(* Logix 5000 project; controller DUNEW2PLC1 vendor 1 type 14 code 221 rev 33.11; software revision 33.00; part 2 of 4 *)
(* tags used below, declared in another part *)
   LatchingTimeoutCounter : COUNTER;   // When you enter state 6 or 7, start counting seconds
   TimeoutTimer1 : TIMER;
   TimeoutTimer2 : TIMER;
   accel_xy : REAL;   // Tangential acceleration of the winding head in xy-plane
   ACTUATOR_POS : DINT;
   ALL_EOT_GOOD : BOOL;
   APA_IS_VERTICAL : BOOL;
   blink_off : TIMER;
   blink_on : TIMER;
   ERROR_CODE : DINT;
   FRAME_LOC_FT_BTM : BOOL;
   FRAME_LOC_FT_MID : BOOL;
   FRAME_LOC_FT_TOP : BOOL;
   FRAME_LOC_HD_BTM : BOOL;
   FRAME_LOC_HD_MID : BOOL;
   FRAME_LOC_HD_TOP : BOOL;
   HEAD_POS : DINT;
   INIT_DONE : BOOL;
   MACHINE_SW_STAT : BOOL[32];
   MAS : BOOL;   // Motion Axis Stop
   MASTER_Z_GO : BOOL;
   MCCD_X_Y_Axis : MOTION_INSTRUCTION;
   MCCD_X_Y_Axis1 : MOTION_INSTRUCTION;
   MINUS_X_EOT : BOOL;
   MINUS_Y_EOT : BOOL;
   MOVE_TYPE : INT;   // 0 = No Move 1 = XY JOG 2 = XY Plane Move 3 = Z JOG 4 = Z Axis Move 5 = Toggle Latch Actuator 6 = Home the Latch Actuator
   NEXTSTATE : DINT;
   PLUS_X_EOT : BOOL;
   PLUS_Y_EOT : BOOL;
   ResetPB : BOOL;
   Safety_Tripped_S : BOOL;
   SLS_speed : DINT;
   speed_regulator_switch : BOOL;   // This is our "enable safe speed" switch, repurposed to switch the speed regulator
   STATE : DINT;   // CURRENT State Machine State
   T01 : TIMER;
   tension : ALIAS FOR Local:4:I.Ch01.Data;   // wire tension (N)
   TENSION_ON_SWITCH : BOOL;
   v_xy : REAL;   // velocity of winding head in xy plane
   v_xyz : REAL;   // Velocity of winding head in xyz space
   wire_break_proxy : BOOL;
   wire_break_tension : REAL;
   X_axis : AXIS_CIP_DRIVE;
   X_Axis_SLS : SAFELY_LIMITED_SPEED;
   X_DIR : DINT;
   X_PARKED : BOOL;
   X_POSITION : ALIAS FOR POSITION[0,0];
   X_SPEED : REAL;
   X_XFER_OK : BOOL;   // If at the head, check head support arms. Same for foot
   X_Y : COORDINATE_SYSTEM;
   XY_ACCELERATION : REAL;   // Maximum positive acceleration for position move.
   XY_DECELERATION : REAL;   // Maximum negative acceleration for position move.
   XY_DECELERATION_SLS : REAL;
   XY_SPEED : REAL;   // Maximum velocity for position move.
   XY_SPEED_REQ : REAL;   // XY Requested speed copy of XY_Speed to be used for MCLM and MCCD in MoveXY
   Y_axis : AXIS_CIP_DRIVE;
   Y_DIR : DINT;
   Y_MOUNT_XFER_OK : BOOL;
   Y_POSITION : ALIAS FOR POSITION[0,1];
   Y_SPEED : REAL;
   Y_XFER_OK : BOOL;
   Y_Xfer_Window_Btm : BOOL;
   Y_Xfer_Window_Mid : BOOL;
   Y_Xfer_Window_Top : BOOL;
   Z_axis : AXIS_CIP_DRIVE;
   Z_EOT : BOOL;
   Z_EXTENDED : BOOL;
   Z_FIXED_LATCHED : BOOL;
   Z_FIXED_PRESENT : BOOL;
   Z_RETRACTED : BOOL;
   Z_STAGE_LATCHED : BOOL;
   Z_STAGE_PRESENT : BOOL;   // Winding head is on the Z-arm
(* Latch_UnLatch_State_6_7_8, continued *)

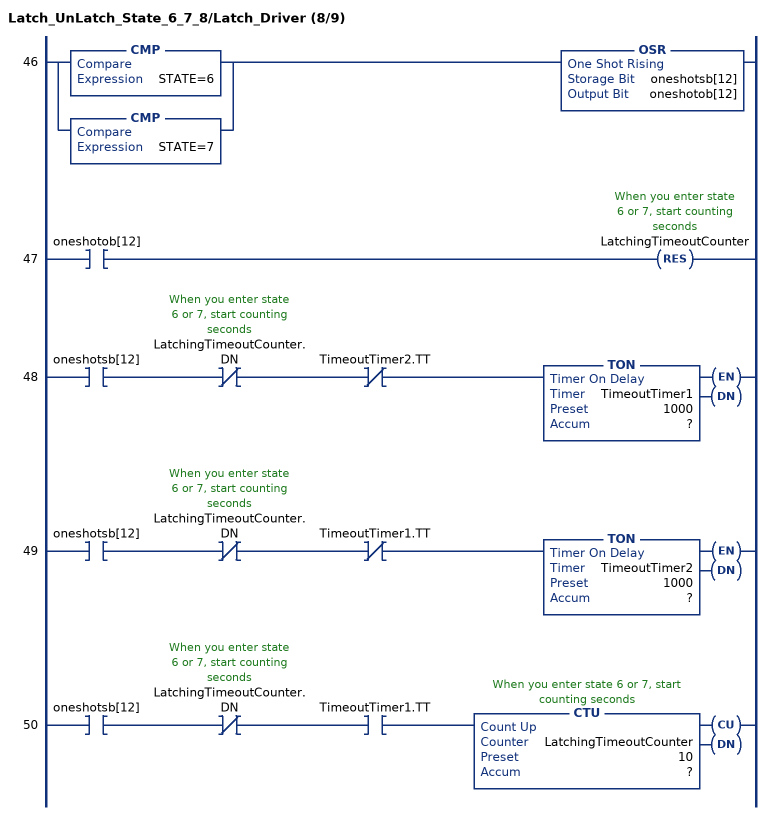
   [picture p24: Latch_UnLatch_State_6_7_8/Latch_Driver rungs 46-50]
   46: [CMP(STATE=6) ,CMP(STATE=7) ]OSR(oneshotsb[12],oneshotob[12]);
   47: XIC(oneshotob[12])RES(LatchingTimeoutCounter);
   48: XIC(oneshotsb[12])XIO(LatchingTimeoutCounter.DN)XIO(TimeoutTimer2.TT)TON(TimeoutTimer1,?,?);
   49: XIC(oneshotsb[12])XIO(LatchingTimeoutCounter.DN)XIO(TimeoutTimer1.TT)TON(TimeoutTimer2,?,?);
   50: XIC(oneshotsb[12])XIO(LatchingTimeoutCounter.DN)XIC(TimeoutTimer1.TT)CTU(LatchingTimeoutCounter,?,?);
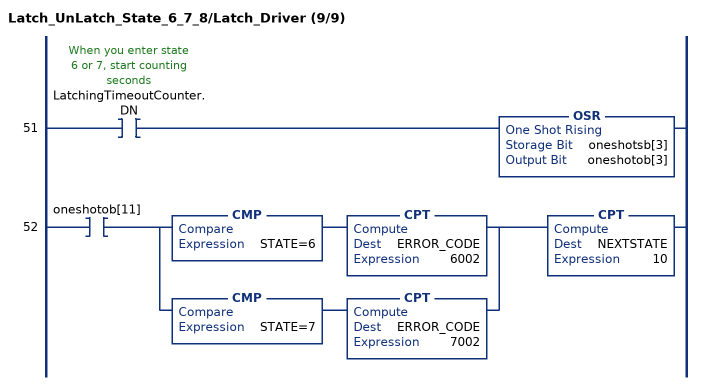
   51: XIC(LatchingTimeoutCounter.DN)OSR(oneshotsb[3],oneshotob[3]);
   52: XIC(oneshotob[11])[CMP(STATE=6) CPT(ERROR_CODE,6002) ,CMP(STATE=7) CPT(ERROR_CODE,7002) ]CPT(NEXTSTATE,10);
END_ROUTINE
END_PROGRAM

PROGRAM MainProgram   (* main routine MainRoutine *)
VAR
   Current_x : REAL := 0.0057; {access Read Only}
   Current_y : DINT; {access Read Only}
   oneshotob : BOOL[32];
   oneshotsb : BOOL[32] := ([4] := 1, [7] := 1);
   STATE2_IND : BOOL; {access Read Only}
   STATE3_IND : BOOL; {access Read Only}
   X_AXIS_STAT : MOTION_INSTRUCTION[32] := ([0].FLAGS := 33554432, [1].FLAGS := 33554432, [2].FLAGS := 33554432);
   XY_AXIS_STAT : MOTION_INSTRUCTION[32] := ([0].FLAGS := 33554432, [1].FLAGS := 33554432, [2].FLAGS := 536870912, [2].DN := 1, [3].FLAGS := 536870912, [3].DN := 1, [4].FLAGS := 704643072, [4].DN := 1, [4].PC := 1, [5].FLAGS := 704643072, [5].DN := 1, [5].PC := 1, [6].FLAGS := 33554432);
   XY_POS_LOCK_STAT : BOOL; {access Read Only}
   XY_SERVO_ON : BOOL; {access Read Only}
   Y_AXIS_STAT : MOTION_INSTRUCTION[32] := ([0].FLAGS := 33554432, [1].FLAGS := 33554432, [2].FLAGS := 33554432);
   Z_RETRACTED_1A : BOOL := 1; {access Read Only}
   Z_RETRACTED_1B : BOOL := 1; {access Read Only}
   Z_RETRACTED_2A : BOOL := 1; {access Read Only}
   Z_RETRACTED_2B : BOOL := 1; {access Read Only}
END_VAR

ROUTINE MainRoutine   (* ladder *)
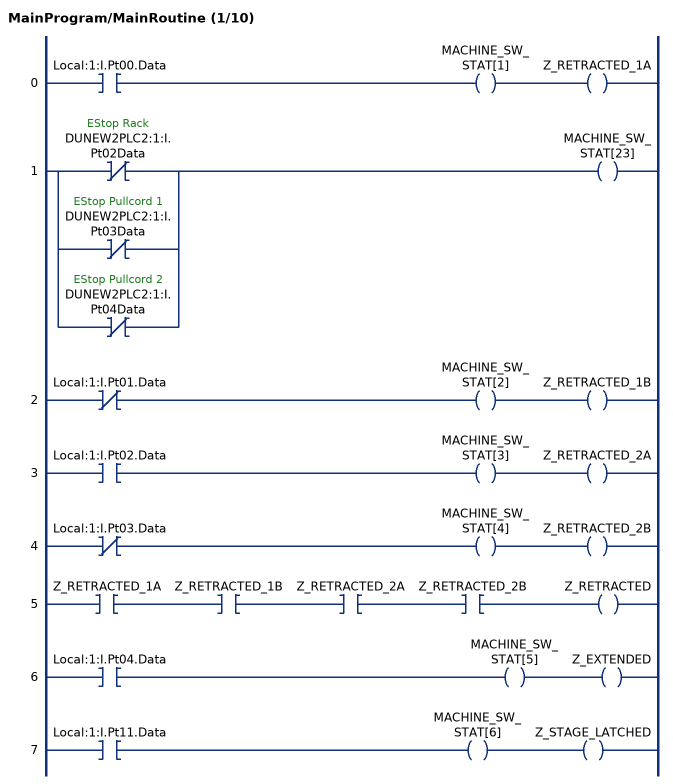
   0: XIC(Local:1:I.Pt00.Data)OTE(MACHINE_SW_STAT[1])OTE(Z_RETRACTED_1A);
   1: [XIO(DUNEW2PLC2:1:I.Pt02Data) ,[XIO(DUNEW2PLC2:1:I.Pt03Data) ,XIO(DUNEW2PLC2:1:I.Pt04Data) ] ]OTE(MACHINE_SW_STAT[23]);
   2: XIO(Local:1:I.Pt01.Data)OTE(MACHINE_SW_STAT[2])OTE(Z_RETRACTED_1B);
   3: XIC(Local:1:I.Pt02.Data)OTE(MACHINE_SW_STAT[3])OTE(Z_RETRACTED_2A);
   4: XIO(Local:1:I.Pt03.Data)OTE(MACHINE_SW_STAT[4])OTE(Z_RETRACTED_2B);
   5: XIC(Z_RETRACTED_1A)XIC(Z_RETRACTED_1B)XIC(Z_RETRACTED_2A)XIC(Z_RETRACTED_2B)OTE(Z_RETRACTED);
   6: XIC(Local:1:I.Pt04.Data)OTE(MACHINE_SW_STAT[5])OTE(Z_EXTENDED);
   7: XIC(Local:1:I.Pt11.Data)OTE(MACHINE_SW_STAT[6])OTE(Z_STAGE_LATCHED);
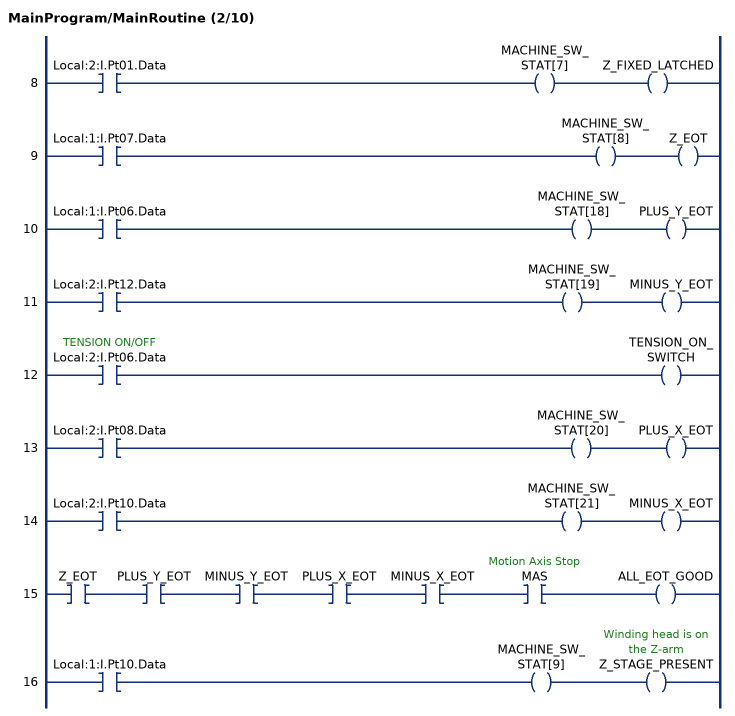
   8: XIC(Local:2:I.Pt01.Data)OTE(MACHINE_SW_STAT[7])OTE(Z_FIXED_LATCHED);
   9: XIC(Local:1:I.Pt07.Data)OTE(MACHINE_SW_STAT[8])OTE(Z_EOT);
   10: XIC(Local:1:I.Pt06.Data)OTE(MACHINE_SW_STAT[18])OTE(PLUS_Y_EOT);
   11: XIC(Local:2:I.Pt12.Data)OTE(MACHINE_SW_STAT[19])OTE(MINUS_Y_EOT);
   12: XIC(Local:2:I.Pt06.Data)OTE(TENSION_ON_SWITCH);
   13: XIC(Local:2:I.Pt08.Data)OTE(MACHINE_SW_STAT[20])OTE(PLUS_X_EOT);
   14: XIC(Local:2:I.Pt10.Data)OTE(MACHINE_SW_STAT[21])OTE(MINUS_X_EOT);
   15: XIC(Z_EOT)XIC(PLUS_Y_EOT)XIC(MINUS_Y_EOT)XIC(PLUS_X_EOT)XIC(MINUS_X_EOT)XIC(MAS)OTE(ALL_EOT_GOOD);
   16: XIC(Local:1:I.Pt10.Data)OTE(MACHINE_SW_STAT[9])OTE(Z_STAGE_PRESENT);
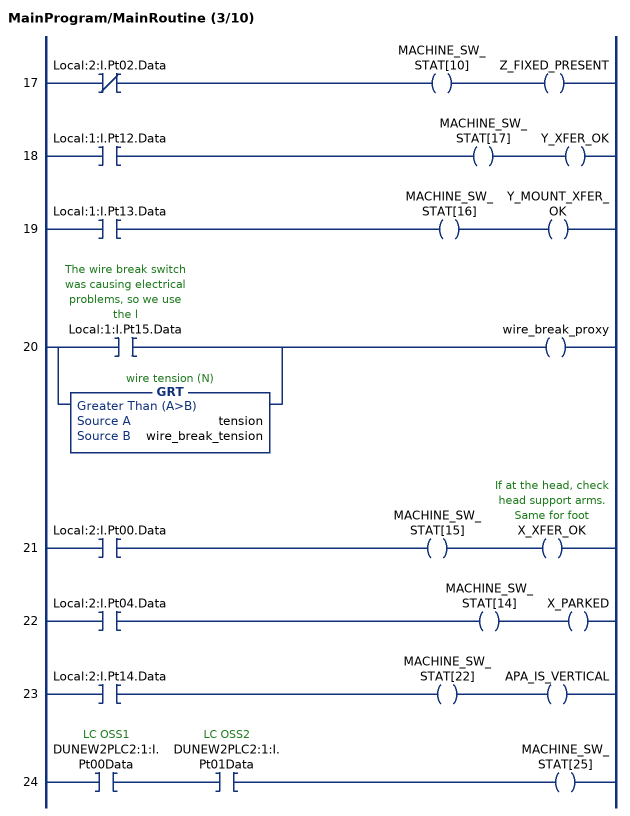
   17: XIO(Local:2:I.Pt02.Data)OTE(MACHINE_SW_STAT[10])OTE(Z_FIXED_PRESENT);
   18: XIC(Local:1:I.Pt12.Data)OTE(MACHINE_SW_STAT[17])OTE(Y_XFER_OK);
   19: XIC(Local:1:I.Pt13.Data)OTE(MACHINE_SW_STAT[16])OTE(Y_MOUNT_XFER_OK);
   20: [XIC(Local:1:I.Pt15.Data) ,GRT(tension,wire_break_tension) ]OTE(wire_break_proxy);
   21: XIC(Local:2:I.Pt00.Data)OTE(MACHINE_SW_STAT[15])OTE(X_XFER_OK);
   22: XIC(Local:2:I.Pt04.Data)OTE(MACHINE_SW_STAT[14])OTE(X_PARKED);
   23: XIC(Local:2:I.Pt14.Data)OTE(MACHINE_SW_STAT[22])OTE(APA_IS_VERTICAL);
   24: XIC(DUNEW2PLC2:1:I.Pt00Data)XIC(DUNEW2PLC2:1:I.Pt01Data)OTE(MACHINE_SW_STAT[25]);
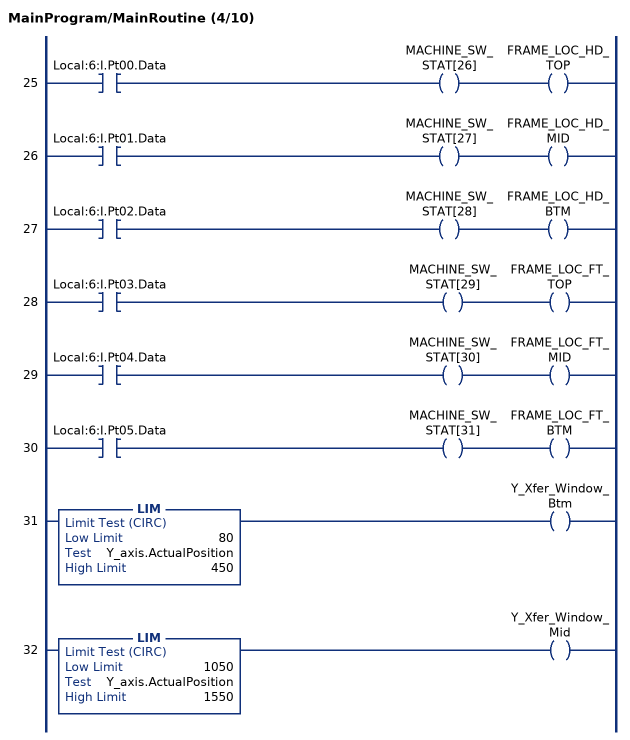
   25: XIC(Local:6:I.Pt00.Data)OTE(MACHINE_SW_STAT[26])OTE(FRAME_LOC_HD_TOP);
   26: XIC(Local:6:I.Pt01.Data)OTE(MACHINE_SW_STAT[27])OTE(FRAME_LOC_HD_MID);
   27: XIC(Local:6:I.Pt02.Data)OTE(MACHINE_SW_STAT[28])OTE(FRAME_LOC_HD_BTM);
   28: XIC(Local:6:I.Pt03.Data)OTE(MACHINE_SW_STAT[29])OTE(FRAME_LOC_FT_TOP);
   29: XIC(Local:6:I.Pt04.Data)OTE(MACHINE_SW_STAT[30])OTE(FRAME_LOC_FT_MID);
   30: XIC(Local:6:I.Pt05.Data)OTE(MACHINE_SW_STAT[31])OTE(FRAME_LOC_FT_BTM);
   31: LIM(80,Y_axis.ActualPosition,450)OTE(Y_Xfer_Window_Btm);
   32: LIM(1050,Y_axis.ActualPosition,1550)OTE(Y_Xfer_Window_Mid);
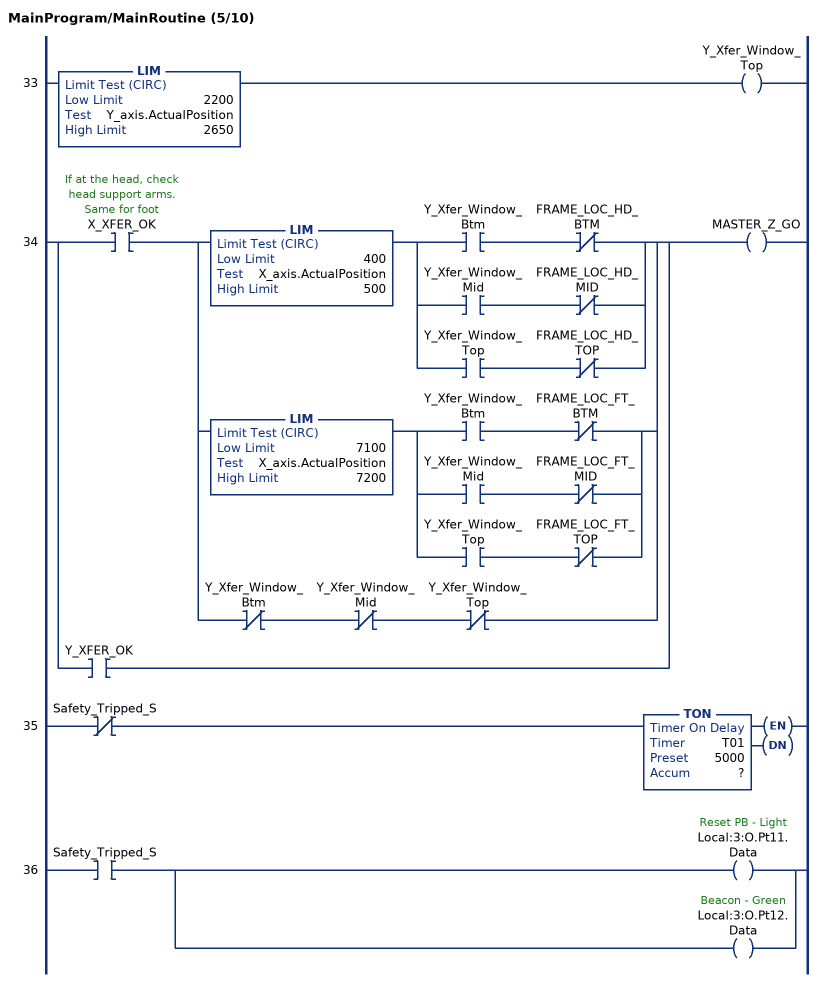
   33: LIM(2200,Y_axis.ActualPosition,2650)OTE(Y_Xfer_Window_Top);
   34: [XIC(X_XFER_OK) [LIM(400,X_axis.ActualPosition,500) [XIC(Y_Xfer_Window_Btm) XIO(FRAME_LOC_HD_BTM) ,XIC(Y_Xfer_Window_Mid) XIO(FRAME_LOC_HD_MID) ,XIC(Y_Xfer_Window_Top) XIO(FRAME_LOC_HD_TOP) ] ,LIM(7100,X_axis.ActualPosition,7200) [XIC(Y_Xfer_Window_Btm) XIO(FRAME_LOC_FT_BTM) ,XIC(Y_Xfer_Window_Mid) XIO(FRAME_LOC_FT_MID) ,XIC(Y_Xfer_Window_Top) XIO(FRAME_LOC_FT_TOP) ] ,XIO(Y_Xfer_Window_Btm) XIO(Y_Xfer_Window_Mid) XIO(Y_Xfer_Window_Top) ] ,XIC(Y_XFER_OK) ]OTE(MASTER_Z_GO);
   35: XIO(Safety_Tripped_S)TON(T01,?,?);
   36: XIC(Safety_Tripped_S)[OTE(Local:3:O.Pt11.Data) ,OTE(Local:3:O.Pt12.Data) ];
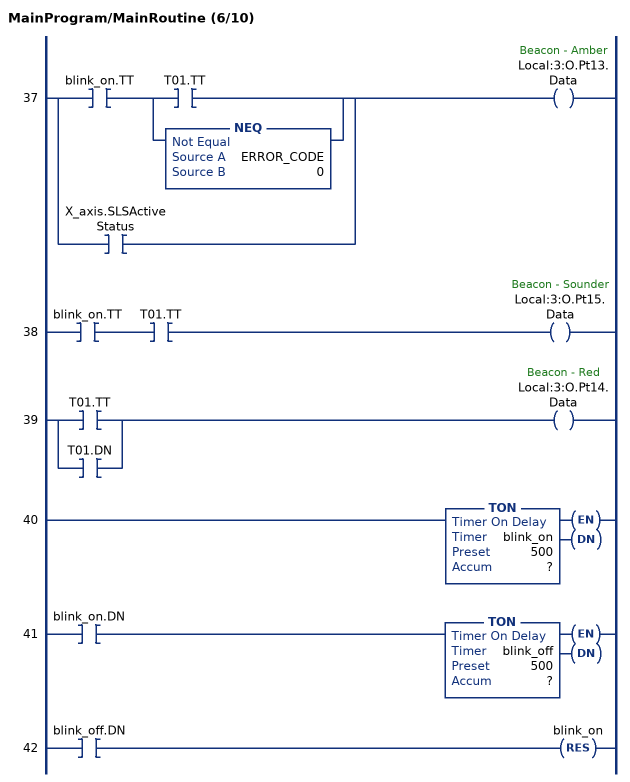
   37: [XIC(blink_on.TT) [XIC(T01.TT) ,NEQ(ERROR_CODE,0) ] ,XIC(X_axis.SLSActiveStatus) ]OTE(Local:3:O.Pt13.Data);
   38: XIC(blink_on.TT)XIC(T01.TT)OTE(Local:3:O.Pt15.Data);
   39: [XIC(T01.TT) ,XIC(T01.DN) ]OTE(Local:3:O.Pt14.Data);
   40: TON(blink_on,?,?);
   41: XIC(blink_on.DN)TON(blink_off,?,?);
   42: XIC(blink_off.DN)RES(blink_on);
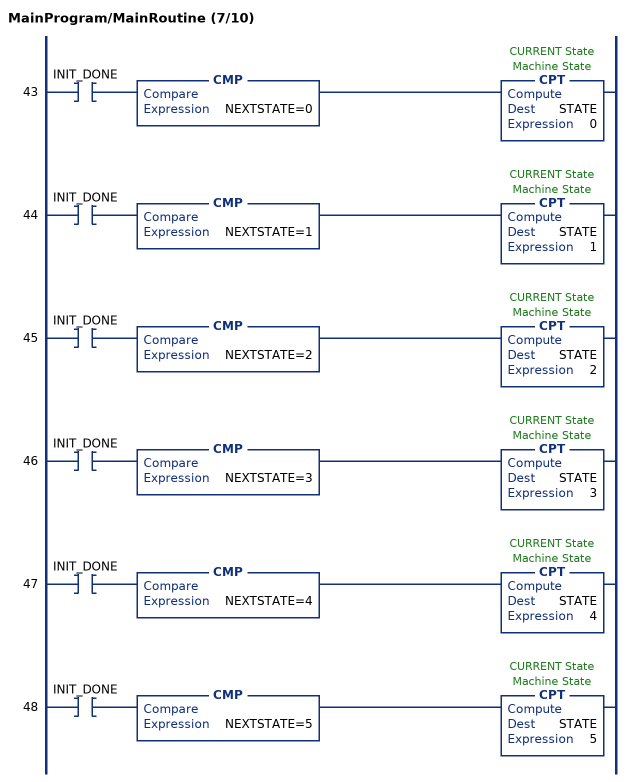
   43: XIC(INIT_DONE)CMP(NEXTSTATE=0)CPT(STATE,0);
   44: XIC(INIT_DONE)CMP(NEXTSTATE=1)CPT(STATE,1);
   45: XIC(INIT_DONE)CMP(NEXTSTATE=2)CPT(STATE,2);
   46: XIC(INIT_DONE)CMP(NEXTSTATE=3)CPT(STATE,3);
   47: XIC(INIT_DONE)CMP(NEXTSTATE=4)CPT(STATE,4);
   48: XIC(INIT_DONE)CMP(NEXTSTATE=5)CPT(STATE,5);
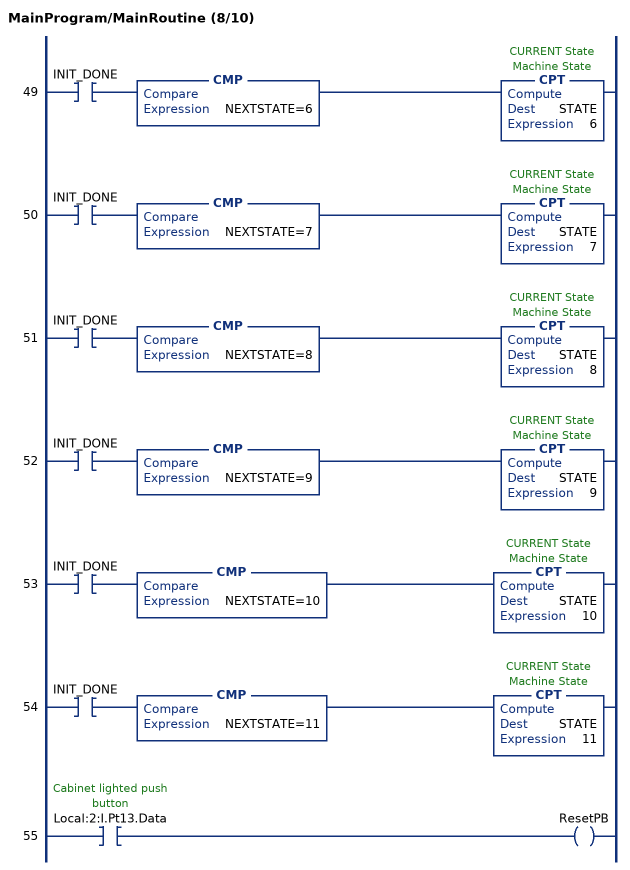
   49: XIC(INIT_DONE)CMP(NEXTSTATE=6)CPT(STATE,6);
   50: XIC(INIT_DONE)CMP(NEXTSTATE=7)CPT(STATE,7);
   51: XIC(INIT_DONE)CMP(NEXTSTATE=8)CPT(STATE,8);
   52: XIC(INIT_DONE)CMP(NEXTSTATE=9)CPT(STATE,9);
   53: XIC(INIT_DONE)CMP(NEXTSTATE=10)CPT(STATE,10);
   54: XIC(INIT_DONE)CMP(NEXTSTATE=11)CPT(STATE,11);
   55: XIC(Local:2:I.Pt13.Data)OTE(ResetPB);
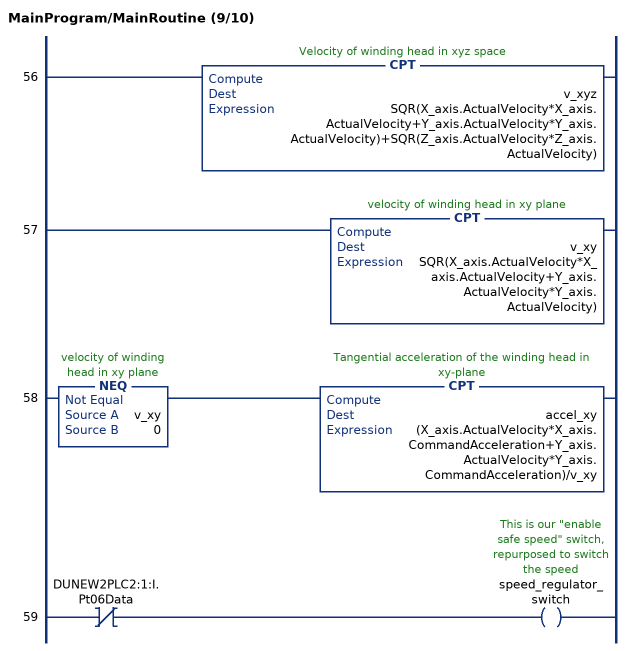
   56: CPT(v_xyz,SQR(X_axis.ActualVelocity*X_axis.ActualVelocity+Y_axis.ActualVelocity*Y_axis.ActualVelocity)+SQR(Z_axis.ActualVelocity*Z_axis.ActualVelocity));
   57: CPT(v_xy,SQR(X_axis.ActualVelocity*X_axis.ActualVelocity+Y_axis.ActualVelocity*Y_axis.ActualVelocity));
   58: NEQ(v_xy,0)CPT(accel_xy,(X_axis.ActualVelocity*X_axis.CommandAcceleration+Y_axis.ActualVelocity*Y_axis.CommandAcceleration)/v_xy);
   59: XIO(DUNEW2PLC2:1:I.Pt06Data)OTE(speed_regulator_switch);
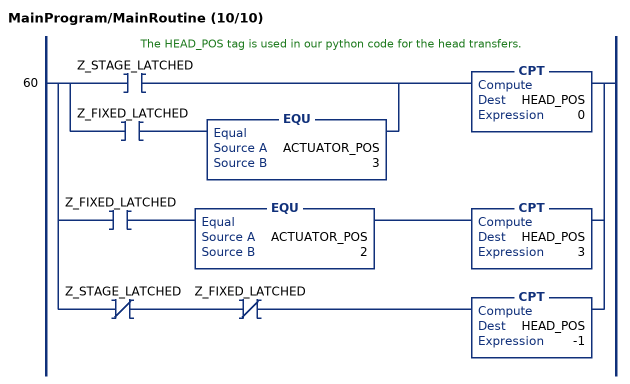
   // The HEAD_POS tag is used in our python code for the head transfers.
   60: [[XIC(Z_STAGE_LATCHED) ,XIC(Z_FIXED_LATCHED) EQU(ACTUATOR_POS,3) ] CPT(HEAD_POS,0) ,XIC(Z_FIXED_LATCHED) EQU(ACTUATOR_POS,2) CPT(HEAD_POS,3) ,XIO(Z_STAGE_LATCHED) XIO(Z_FIXED_LATCHED) CPT(HEAD_POS,-1) ];
END_ROUTINE

ROUTINE MoveXY   (* ladder *)
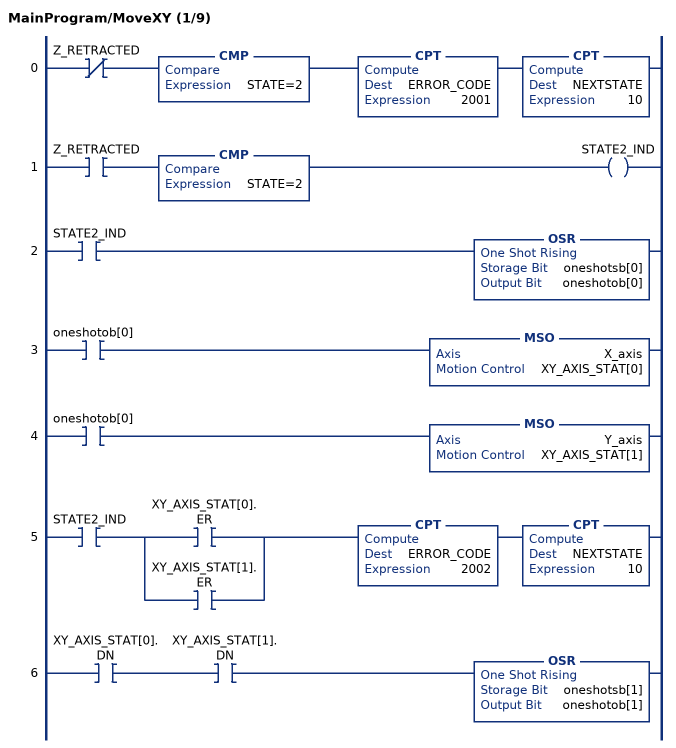
   0: XIO(Z_RETRACTED)CMP(STATE=2)CPT(ERROR_CODE,2001)CPT(NEXTSTATE,10);
   1: XIC(Z_RETRACTED)CMP(STATE=2)OTE(STATE2_IND);
   2: XIC(STATE2_IND)OSR(oneshotsb[0],oneshotob[0]);
   3: XIC(oneshotob[0])MSO(X_axis,XY_AXIS_STAT[0]);
   4: XIC(oneshotob[0])MSO(Y_axis,XY_AXIS_STAT[1]);
   5: XIC(STATE2_IND)[XIC(XY_AXIS_STAT[0].ER) ,XIC(XY_AXIS_STAT[1].ER) ]CPT(ERROR_CODE,2002)CPT(NEXTSTATE,10);
   6: XIC(XY_AXIS_STAT[0].DN)XIC(XY_AXIS_STAT[1].DN)OSR(oneshotsb[1],oneshotob[1]);
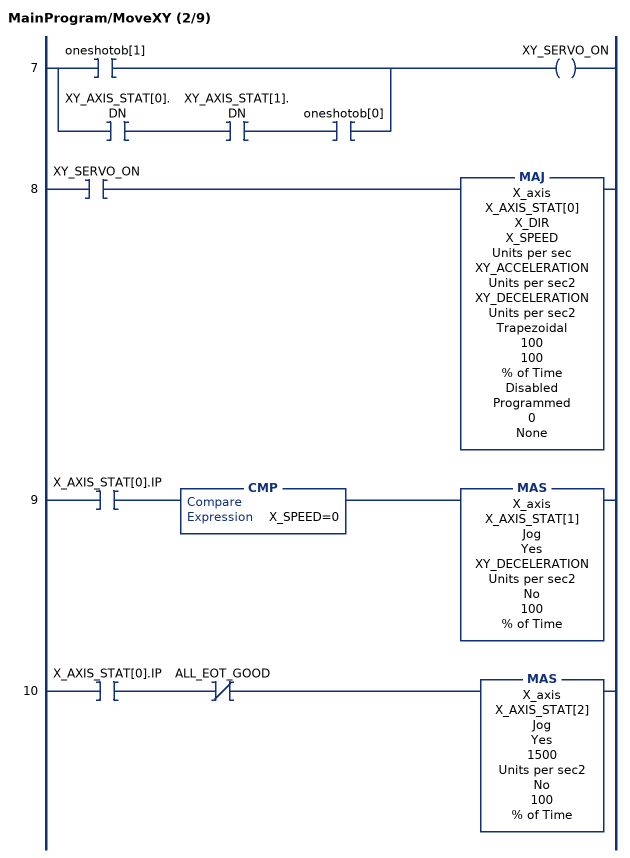
   7: [XIC(oneshotob[1]) ,XIC(XY_AXIS_STAT[0].DN) XIC(XY_AXIS_STAT[1].DN) XIC(oneshotob[0]) ]OTE(XY_SERVO_ON);
   8: XIC(XY_SERVO_ON)MAJ(X_axis,X_AXIS_STAT[0],X_DIR,X_SPEED,Units per sec,XY_ACCELERATION,Units per sec2,XY_DECELERATION,Units per sec2,Trapezoidal,100,100,% of Time,Disabled,Programmed,0,None);
   9: XIC(X_AXIS_STAT[0].IP)CMP(X_SPEED=0)MAS(X_axis,X_AXIS_STAT[1],Jog,Yes,XY_DECELERATION,Units per sec2,No,100,% of Time);
   10: XIC(X_AXIS_STAT[0].IP)XIO(ALL_EOT_GOOD)MAS(X_axis,X_AXIS_STAT[2],Jog,Yes,1500,Units per sec2,No,100,% of Time);
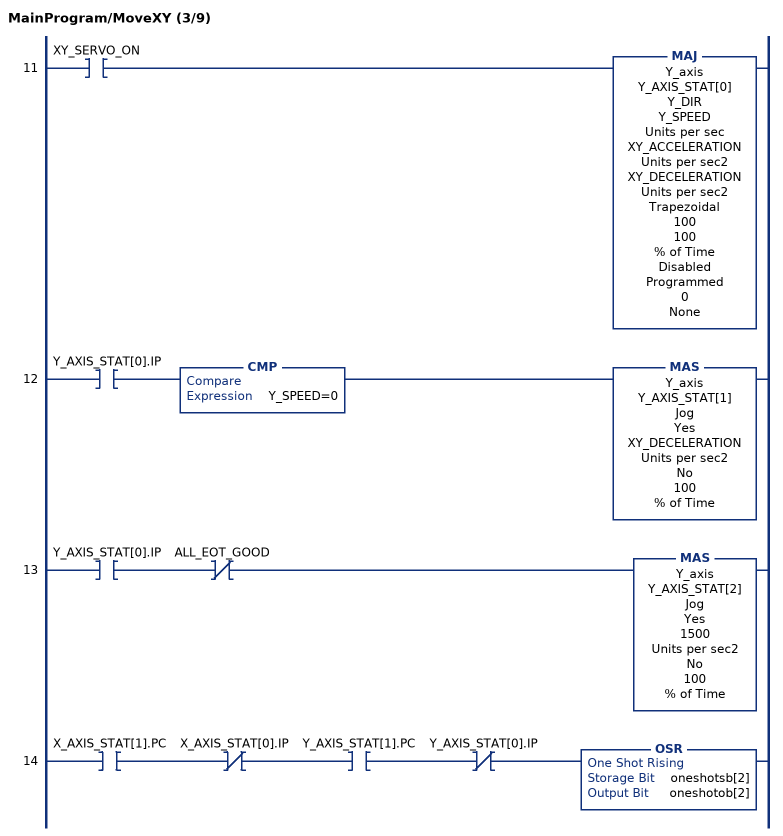
   11: XIC(XY_SERVO_ON)MAJ(Y_axis,Y_AXIS_STAT[0],Y_DIR,Y_SPEED,Units per sec,XY_ACCELERATION,Units per sec2,XY_DECELERATION,Units per sec2,Trapezoidal,100,100,% of Time,Disabled,Programmed,0,None);
   12: XIC(Y_AXIS_STAT[0].IP)CMP(Y_SPEED=0)MAS(Y_axis,Y_AXIS_STAT[1],Jog,Yes,XY_DECELERATION,Units per sec2,No,100,% of Time);
   13: XIC(Y_AXIS_STAT[0].IP)XIO(ALL_EOT_GOOD)MAS(Y_axis,Y_AXIS_STAT[2],Jog,Yes,1500,Units per sec2,No,100,% of Time);
   14: XIC(X_AXIS_STAT[1].PC)XIO(X_AXIS_STAT[0].IP)XIC(Y_AXIS_STAT[1].PC)XIO(Y_AXIS_STAT[0].IP)OSR(oneshotsb[2],oneshotob[2]);
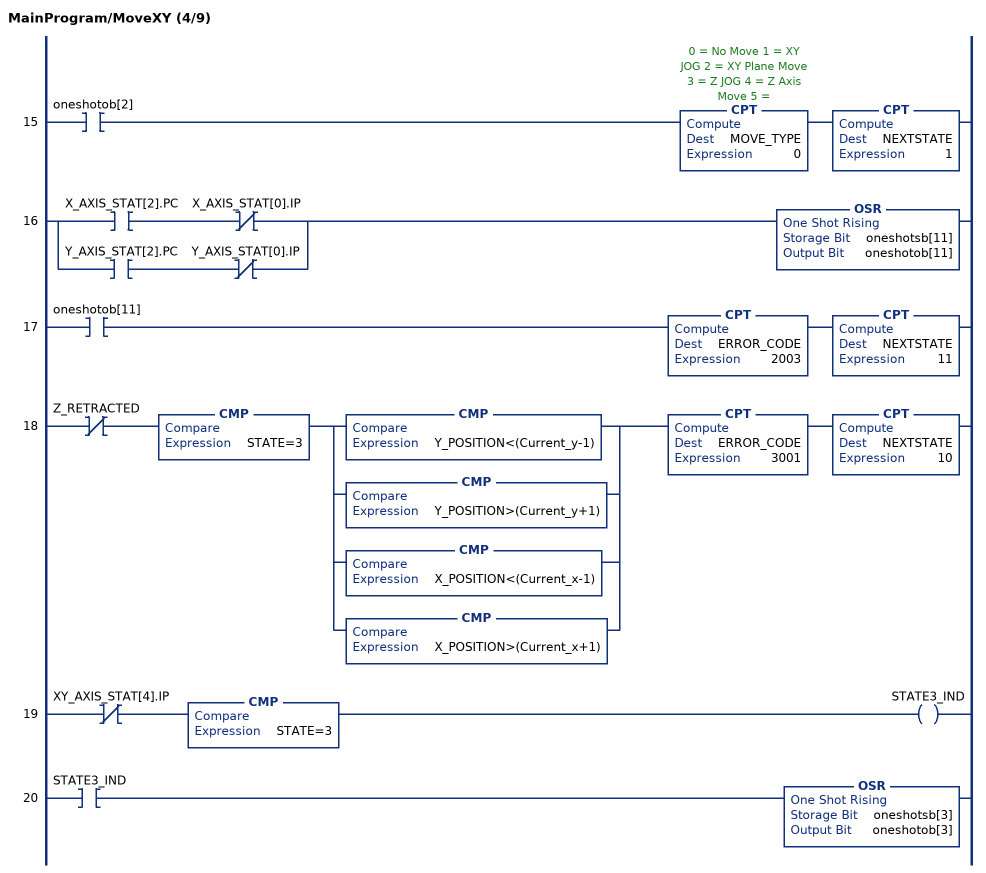
   15: XIC(oneshotob[2])CPT(MOVE_TYPE,0)CPT(NEXTSTATE,1);
   16: [XIC(X_AXIS_STAT[2].PC) XIO(X_AXIS_STAT[0].IP) ,XIC(Y_AXIS_STAT[2].PC) XIO(Y_AXIS_STAT[0].IP) ]OSR(oneshotsb[11],oneshotob[11]);
   17: XIC(oneshotob[11])CPT(ERROR_CODE,2003)CPT(NEXTSTATE,11);
   18: XIO(Z_RETRACTED)CMP(STATE=3)[CMP(Y_POSITION<(Current_y-1)) ,CMP(Y_POSITION>(Current_y+1)) ,CMP(X_POSITION<(Current_x-1)) ,CMP(X_POSITION>(Current_x+1)) ]CPT(ERROR_CODE,3001)CPT(NEXTSTATE,10);
   19: XIO(XY_AXIS_STAT[4].IP)CMP(STATE=3)OTE(STATE3_IND);
   20: XIC(STATE3_IND)OSR(oneshotsb[3],oneshotob[3]);
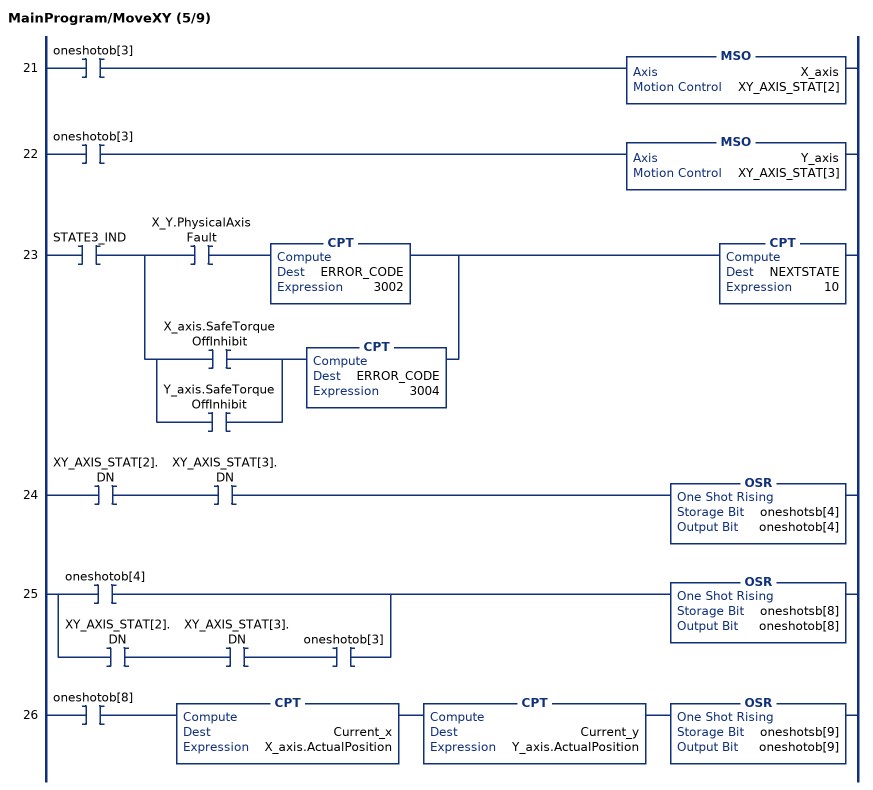
   21: XIC(oneshotob[3])MSO(X_axis,XY_AXIS_STAT[2]);
   22: XIC(oneshotob[3])MSO(Y_axis,XY_AXIS_STAT[3]);
   23: XIC(STATE3_IND)[XIC(X_Y.PhysicalAxisFault) CPT(ERROR_CODE,3002) ,[XIC(X_axis.SafeTorqueOffInhibit) ,XIC(Y_axis.SafeTorqueOffInhibit) ] CPT(ERROR_CODE,3004) ]CPT(NEXTSTATE,10);
   24: XIC(XY_AXIS_STAT[2].DN)XIC(XY_AXIS_STAT[3].DN)OSR(oneshotsb[4],oneshotob[4]);
   25: [XIC(oneshotob[4]) ,XIC(XY_AXIS_STAT[2].DN) XIC(XY_AXIS_STAT[3].DN) XIC(oneshotob[3]) ]OSR(oneshotsb[8],oneshotob[8]);
   26: XIC(oneshotob[8])CPT(Current_x,X_axis.ActualPosition)CPT(Current_y,Y_axis.ActualPosition)OSR(oneshotsb[9],oneshotob[9]);
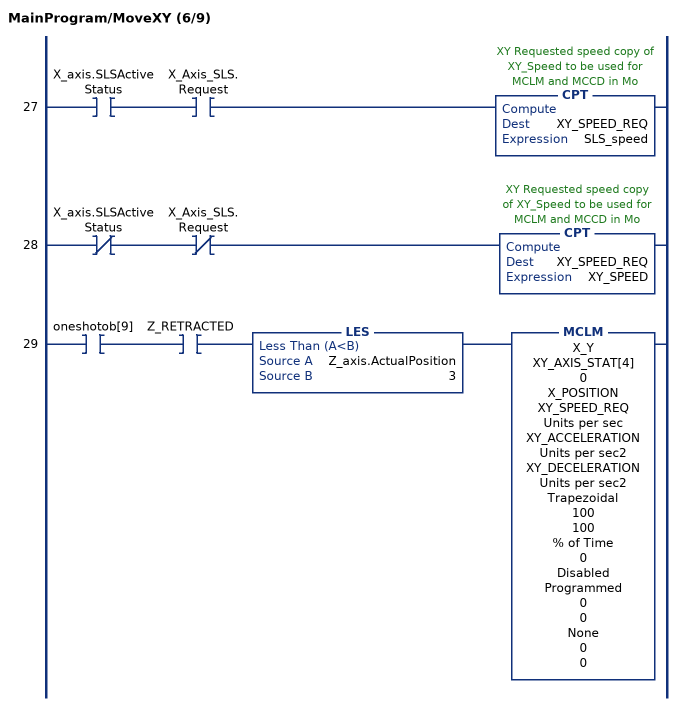
   27: XIC(X_axis.SLSActiveStatus)XIC(X_Axis_SLS.Request)CPT(XY_SPEED_REQ,SLS_speed);
   28: XIO(X_axis.SLSActiveStatus)XIO(X_Axis_SLS.Request)CPT(XY_SPEED_REQ,XY_SPEED);
   29: XIC(oneshotob[9])XIC(Z_RETRACTED)LES(Z_axis.ActualPosition,3)MCLM(X_Y,XY_AXIS_STAT[4],0,X_POSITION,XY_SPEED_REQ,Units per sec,XY_ACCELERATION,Units per sec2,XY_DECELERATION,Units per sec2,Trapezoidal,100,100,% of Time,0,Disabled,Programmed,0,0,None,0,0);
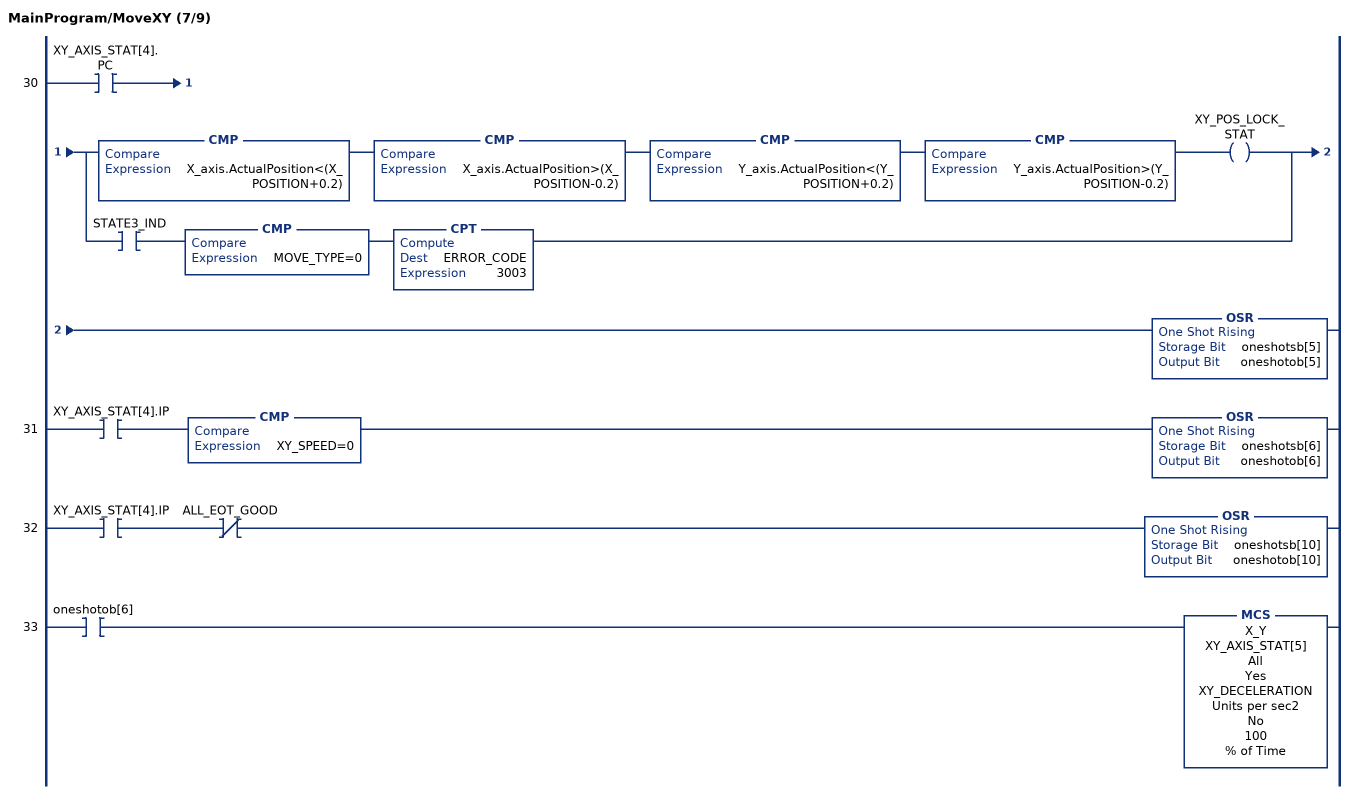
   30: XIC(XY_AXIS_STAT[4].PC)[CMP(X_axis.ActualPosition<(X_POSITION+0.2)) CMP(X_axis.ActualPosition>(X_POSITION-0.2)) CMP(Y_axis.ActualPosition<(Y_POSITION+0.2)) CMP(Y_axis.ActualPosition>(Y_POSITION-0.2)) OTE(XY_POS_LOCK_STAT) ,XIC(STATE3_IND) CMP(MOVE_TYPE=0) CPT(ERROR_CODE,3003) ]OSR(oneshotsb[5],oneshotob[5]);
   31: XIC(XY_AXIS_STAT[4].IP)CMP(XY_SPEED=0)OSR(oneshotsb[6],oneshotob[6]);
   32: XIC(XY_AXIS_STAT[4].IP)XIO(ALL_EOT_GOOD)OSR(oneshotsb[10],oneshotob[10]);
   33: XIC(oneshotob[6])MCS(X_Y,XY_AXIS_STAT[5],All,Yes,XY_DECELERATION,Units per sec2,No,100,% of Time);
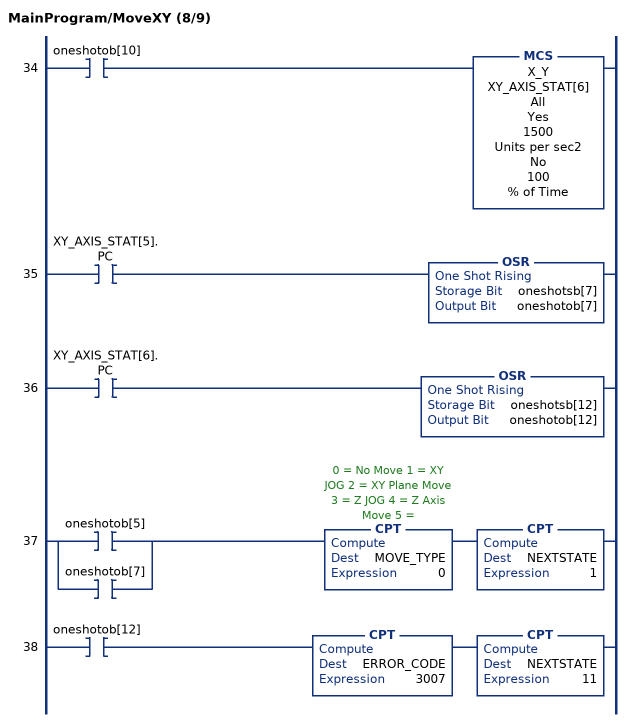
   34: XIC(oneshotob[10])MCS(X_Y,XY_AXIS_STAT[6],All,Yes,1500,Units per sec2,No,100,% of Time);
   35: XIC(XY_AXIS_STAT[5].PC)OSR(oneshotsb[7],oneshotob[7]);
   36: XIC(XY_AXIS_STAT[6].PC)OSR(oneshotsb[12],oneshotob[12]);
   37: [XIC(oneshotob[5]) ,XIC(oneshotob[7]) ]CPT(MOVE_TYPE,0)CPT(NEXTSTATE,1);
   38: XIC(oneshotob[12])CPT(ERROR_CODE,3007)CPT(NEXTSTATE,11);
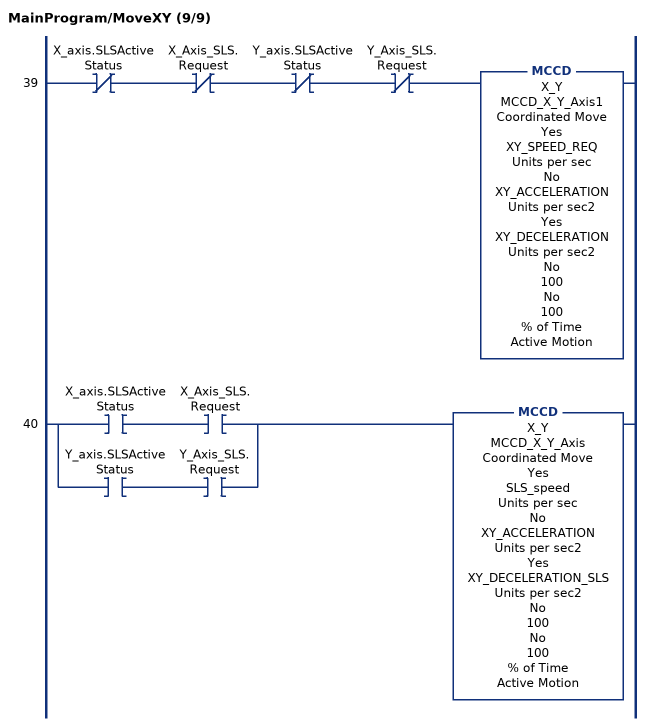
   39: XIO(X_axis.SLSActiveStatus)XIO(X_Axis_SLS.Request)XIO(Y_axis.SLSActiveStatus)XIO(Y_Axis_SLS.Request)MCCD(X_Y,MCCD_X_Y_Axis1,Coordinated Move,Yes,XY_SPEED_REQ,Units per sec,No,XY_ACCELERATION,Units per sec2,Yes,XY_DECELERATION,Units per sec2,No,100,No,100,% of Time,Active Motion);
   40: [XIC(X_axis.SLSActiveStatus) XIC(X_Axis_SLS.Request) ,XIC(Y_axis.SLSActiveStatus) XIC(Y_Axis_SLS.Request) ]MCCD(X_Y,MCCD_X_Y_Axis,Coordinated Move,Yes,SLS_speed,Units per sec,No,XY_ACCELERATION,Units per sec2,Yes,XY_DECELERATION_SLS,Units per sec2,No,100,No,100,% of Time,Active Motion);
END_ROUTINE
END_PROGRAM
